% RSLogix 500 project project 9.RSS, saved by version 8.30.00.16 %
PROJECT "UNTITLED"    % processor: Bul.1763 MicroLogix 1100 Series B %

PROGRAM FILES
  LAD 2 "MAIN"  13 rungs

DATA FILES
  O0 OUTPUT  4 elements
  I1 INPUT  6 elements
  S2 STATUS  66 elements
  B3 BINARY  4 elements
  T4 TIMER  1 elements
  C5 COUNTER  1 elements
  R6 CONTROL  1 elements
  N7 INTEGER  5 elements
  F8 FLOAT  1 elements
  ST9 STRINGS  8 elements

LADDER 2 "MAIN"
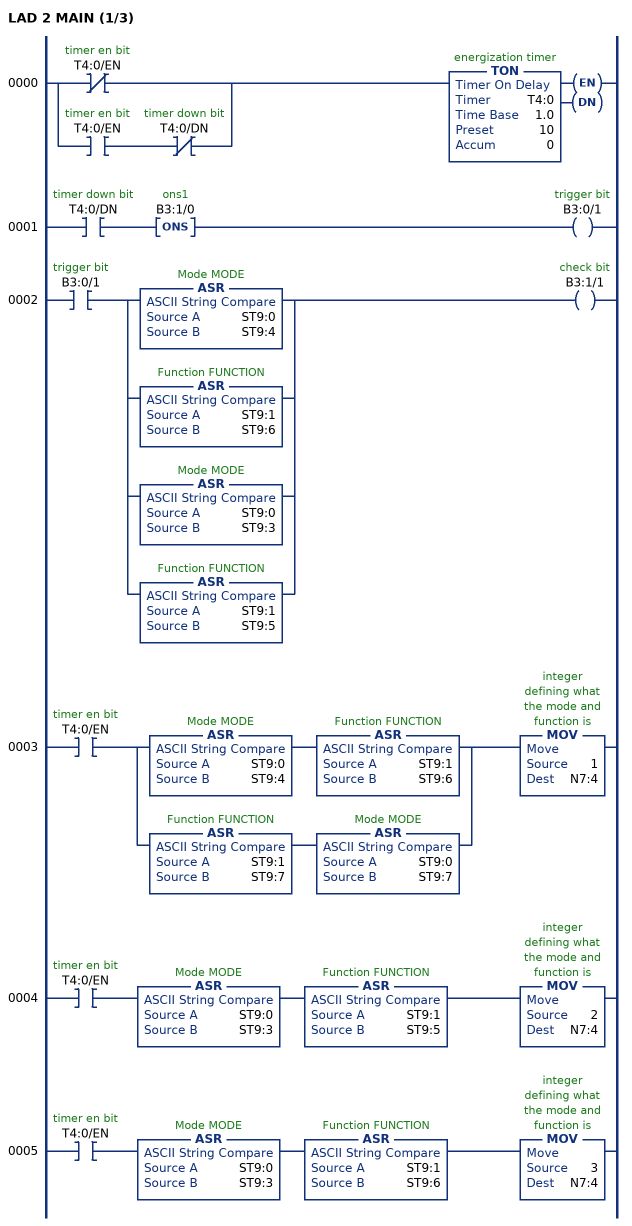
% Rung: 0 %
SOR BST XIO T4:0/EN NXB XIC T4:0/EN XIO T4:0/DN BND TON T4:0 1.0 10 0 EOR
%   T4:0/EN  "timer en bit" %
%   T4:0/DN  "timer down bit" %
%   T4:0  "energization timer" %
% Rung: 1 %
SOR XIC T4:0/DN ONS B3:1/0 OTE B3:0/1 EOR
%   T4:0/DN  "timer down bit" %
%   B3:1/0  "ons1" %
%   B3:0/1  "trigger bit" %
% Rung: 2 %
SOR XIC B3:0/1 BST ASR ST9:0 ST9:4 NXB ASR ST9:1 ST9:6 NXB ASR ST9:0 ST9:3 NXB ASR ST9:1 ST9:5 BND OTE B3:1/1 EOR
%   B3:0/1  "trigger bit" %
%   ST9:0  MODE  "Mode" %
%   ST9:4  "Mode-2" %
%   ST9:1  FUNCTION  "Function" %
%   ST9:6  F2  "F2" %
%   ST9:3  "Mode-1" %
%   ST9:5  F1  "F1" %
%   B3:1/1  "check bit" %
% Rung: 3 %
SOR XIC T4:0/EN BST ASR ST9:0 ST9:4 ASR ST9:1 ST9:6 NXB ASR ST9:1 ST9:7 ASR ST9:0 ST9:7 BND MOV 1 N7:4 EOR
%   T4:0/EN  "timer en bit" %
%   ST9:0  MODE  "Mode" %
%   ST9:4  "Mode-2" %
%   ST9:1  FUNCTION  "Function" %
%   ST9:6  F2  "F2" %
%   N7:4  "integer defining what the mode and function is" %
% Rung: 4 %
SOR XIC T4:0/EN ASR ST9:0 ST9:3 ASR ST9:1 ST9:5 MOV 2 N7:4 EOR
%   T4:0/EN  "timer en bit" %
%   ST9:0  MODE  "Mode" %
%   ST9:3  "Mode-1" %
%   ST9:1  FUNCTION  "Function" %
%   ST9:5  F1  "F1" %
%   N7:4  "integer defining what the mode and function is" %
% Rung: 5 %
SOR XIC T4:0/EN ASR ST9:0 ST9:3 ASR ST9:1 ST9:6 MOV 3 N7:4 EOR
%   T4:0/EN  "timer en bit" %
%   ST9:0  MODE  "Mode" %
%   ST9:3  "Mode-1" %
%   ST9:1  FUNCTION  "Function" %
%   ST9:6  F2  "F2" %
%   N7:4  "integer defining what the mode and function is" %

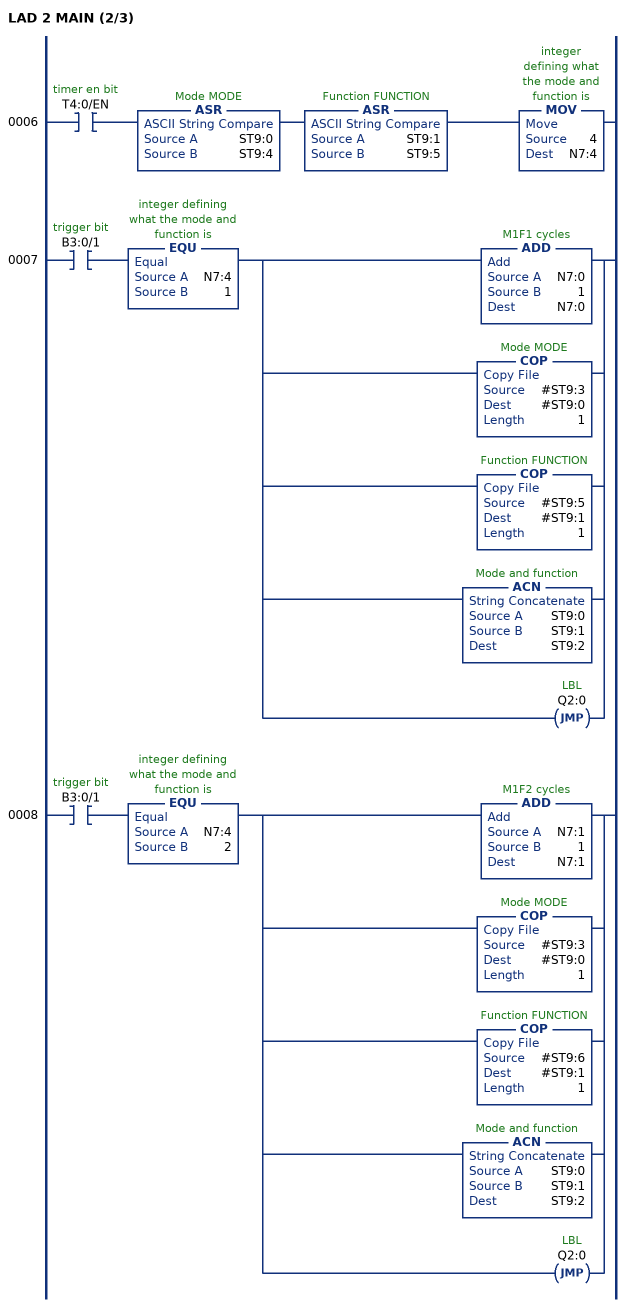
% Rung: 6 %
SOR XIC T4:0/EN ASR ST9:0 ST9:4 ASR ST9:1 ST9:5 MOV 4 N7:4 EOR
%   T4:0/EN  "timer en bit" %
%   ST9:0  MODE  "Mode" %
%   ST9:4  "Mode-2" %
%   ST9:1  FUNCTION  "Function" %
%   ST9:5  F1  "F1" %
%   N7:4  "integer defining what the mode and function is" %
% Rung: 7 %
SOR XIC B3:0/1 EQU N7:4 1 BST ADD N7:0 1 N7:0 NXB COP #ST9:3 #ST9:0 1 NXB COP #ST9:5 #ST9:1 1 NXB ACN ST9:0 ST9:1 ST9:2 NXB JMP Q2:0 BND EOR
%   B3:0/1  "trigger bit" %
%   N7:4  "integer defining what the mode and function is" %
%   N7:0  "M1F1 cycles" %
%   ST9:3  "Mode-1" %
%   ST9:0  MODE  "Mode" %
%   ST9:5  F1  "F1" %
%   ST9:1  FUNCTION  "Function" %
%   ST9:2  "Mode and function" %
%   Q2:0  "LBL" %
% Rung: 8 %
SOR XIC B3:0/1 EQU N7:4 2 BST ADD N7:1 1 N7:1 NXB COP #ST9:3 #ST9:0 1 NXB COP #ST9:6 #ST9:1 1 NXB ACN ST9:0 ST9:1 ST9:2 NXB JMP Q2:0 BND EOR
%   B3:0/1  "trigger bit" %
%   N7:4  "integer defining what the mode and function is" %
%   N7:1  "M1F2 cycles" %
%   ST9:3  "Mode-1" %
%   ST9:0  MODE  "Mode" %
%   ST9:6  F2  "F2" %
%   ST9:1  FUNCTION  "Function" %
%   ST9:2  "Mode and function" %
%   Q2:0  "LBL" %

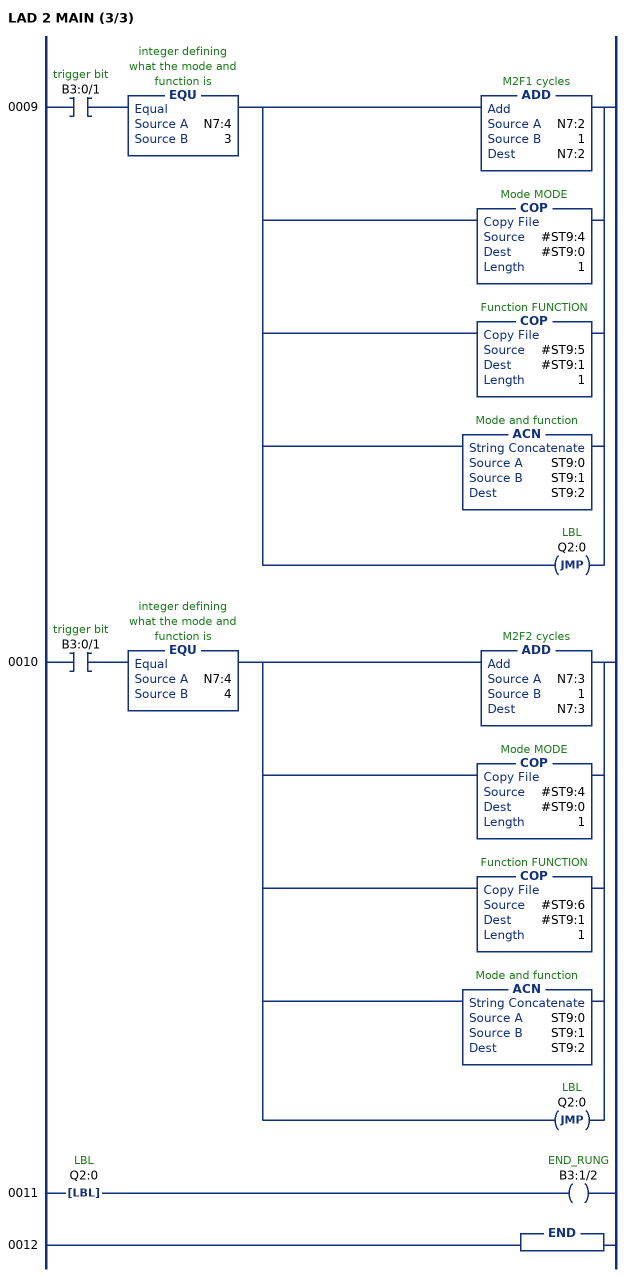
% Rung: 9 %
SOR XIC B3:0/1 EQU N7:4 3 BST ADD N7:2 1 N7:2 NXB COP #ST9:4 #ST9:0 1 NXB COP #ST9:5 #ST9:1 1 NXB ACN ST9:0 ST9:1 ST9:2 NXB JMP Q2:0 BND EOR
%   B3:0/1  "trigger bit" %
%   N7:4  "integer defining what the mode and function is" %
%   N7:2  "M2F1 cycles" %
%   ST9:4  "Mode-2" %
%   ST9:0  MODE  "Mode" %
%   ST9:5  F1  "F1" %
%   ST9:1  FUNCTION  "Function" %
%   ST9:2  "Mode and function" %
%   Q2:0  "LBL" %
% Rung: 10 %
SOR XIC B3:0/1 EQU N7:4 4 BST ADD N7:3 1 N7:3 NXB COP #ST9:4 #ST9:0 1 NXB COP #ST9:6 #ST9:1 1 NXB ACN ST9:0 ST9:1 ST9:2 NXB JMP Q2:0 BND EOR
%   B3:0/1  "trigger bit" %
%   N7:4  "integer defining what the mode and function is" %
%   N7:3  "M2F2 cycles" %
%   ST9:4  "Mode-2" %
%   ST9:0  MODE  "Mode" %
%   ST9:6  F2  "F2" %
%   ST9:1  FUNCTION  "Function" %
%   ST9:2  "Mode and function" %
%   Q2:0  "LBL" %
% Rung: 11 %
SOR LBL Q2:0 OTE B3:1/2 EOR
%   Q2:0  "LBL" %
%   B3:1/2  END_RUNG %
% Rung: 12 %
SOR END EOR

OTHER DOCUMENTED ADDRESSES
  B3:3/0  "toggle bit"
  B3:3/1  "trigger bit"
  Q4:0  "end rung"

DATA TABLE (non-zero values as saved)
DATA T4
% .PRE .ACC %
% T4:0 % 10 0
DATA ST9
% ST9:3 % "Mode-1"
% ST9:4 % "Mode-2"
% ST9:5 % "F1"
% ST9:6 % "F2"
